# EPICS substitutions: src/makeBaseApp/top/pcdsEvrApp/autosaveSrc/autosave__APPNAME_.substitutions
#
# _APPNAME_ substitutions file
#

# Generate iocAdmin autosave request
file autosave_iocAdmin.template
{
	{
		# Hack till msi supports empty substitutions
		_FOOBAR_=_FOOBAR_
	}
}

# Generate EVR autosave request
file autosave_evr.template
{
	{
		# Hack till msi supports empty substitutions
		_FOOBAR_=_FOOBAR_
	}
}
